(* CoDeSys 2.3.9.55 project: AperturaConClave.pro *)
(* Libraries: Standard.lib 2.6.14 11:37:46 *)

(* Global variable list: Global_Variables *)
VAR_GLOBAL

   (* Entradas *)
  (* Botonera de entrada *)
   Ent1:BOOL;
   Ent2:BOOL;
   Ent3:BOOL;
   Ent4:BOOL;
   Cierre:BOOL;


   (* Salidas *)
   CajaAbierta: BOOL;

   (*Claves *)
   Clave1:INT:=1;
  Clave2:INT:=2;
  Clave3:INT:=2;



END_VAR

(* POU PLC_PRG, ST *)
PROGRAM PLC_PRG
VAR
END_VAR
;
END_PROGRAM

(* Visualisation Visu
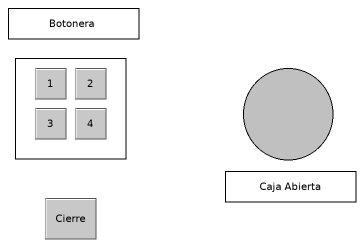
button at (50,130)-(81,161): text "1"; taps Ent1
button at (90,130)-(121,161): text "2"; taps Ent2
button at (50,170)-(81,201): text "3"; taps Ent3
button at (90,170)-(121,201): text "4"; taps Ent4
button at (60,260)-(111,301): text "Cierre"; taps Cierre
rectangle at (23,70)-(154,101): text "Botonera"
ellipse at (258,130)-(348,222): alarm colour if CajaAbierta
rectangle at (240,233)-(371,264): text "Caja Abierta"
1 more shapes without text or variables
*)
